// TIA Portal V16 export
// export: Created 2021-07-12T14:47:19.2126175Z, ExportSetting WithDefaults, DisplayName Totally Integrated Automation Portal, DisplayVersion V16, DisplayName TIA Portal Version Control Interface, DisplayVersion V16, DisplayName TIA Portal Openness, DisplayVersion V16, DisplayName STEP 7 Professional, DisplayVersion V16, DisplayName STEP 7 Safety, DisplayVersion V16, DisplayName WinCC Professional, DisplayVersion V16
TYPE "LSimaHydTO_typeStatusForce"
TITLE = LSimaHydTO_typeStatusForce
// Indicates the status of force control
// stored: IsFailsafeCompliant false
   STRUCT
      ForceLimitingCommand { ExternalWritable := 'False'} : Bool;   // TRUE: Axis is in force limiting mode; FALSE: Axis isn't in force limiting mode/ SimaHyd only
      InLimitation { ExternalWritable := 'False'} : Bool;   // TRUE: Axis is operating at the force limit; FALSE: axis is not operating at the force limit/ SimaHyd only
      InClamping { ExternalWritable := 'False'} : Bool;   // TRUE: Axis is clamped at a fixed stop; FALSE: Axis is not clamped at a fixed stop
      ForceControl { ExternalWritable := 'False'} : Bool;   // TRUE: Axis is in force control mode; FALSE: Axis isn't in force control mode/ SimaHyd only
      TargetForce { ExternalWritable := 'False'} : LReal;   // Target force
      ForceDerivedValue { ExternalWritable := 'False'} : LReal;   // Rate-of-change limiting for the force setpoint
      PreControlValue { ExternalWritable := 'False'} : LReal;   // Force precontrol value
      BalancedForce { ExternalWritable := 'False'} : LReal;   // Force after the balancing filter
      ControlDifference { ExternalWritable := 'False'} : LReal;   // Control error
      ControlOutput { ExternalWritable := 'False'} : LReal;   // Control variable
   END_STRUCT;
END_TYPE
